FUNCTION_BLOCK const_AX_FALSE (* a CONST FALSE for AX Interface *)
  (* Standard: 61499-2 *)
  (* Version 1.0, 2026-08-13, franz, HR Agrartechnik GmbH *)
  PACKAGE adapter::types::unidirectional::AX::constants;
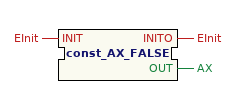
  EVENT_INPUT
    INIT : EInit; (* Initialization Request *)
  END_EVENT
  EVENT_OUTPUT
    INITO : EInit; (* Initialization Confirm *)
  END_EVENT
  PLUGS
    OUT : adapter::types::unidirectional::AX(D1 := FALSE); (* will output FALSE at INIT *)
  END_PLUGS
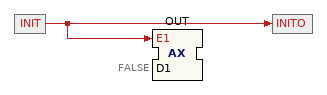
  EVENT_CONNECTIONS
    INIT TO INITO;
    INIT TO OUT.E1;
  END_CONNECTIONS
END_FUNCTION_BLOCK
